// TIA Portal project "ODK_Test" (V14)

(* hardware
DEVICE "OC1"  CPU 1515SP PC
   slot 0: "OC1"  CPU 1515SP PC  6ES7 677-2AAxx-0xB0  V2.0
      slot 124: "Diagbase"  Diagbase  V6.0.4
      slot 125: "OC1"  PC Station 2.0  Station_Manager  V2.1
   slot 1: "CPU1505_v2"  CPU 1505SP  6ES7 672-5DC01-0YA0  V2.0
      slot 3: "CPU display_1"  6ES7591-1BA00-0AA0
   slot 2: "PROFINET onboard_2"  IE General  IE_CP  V2.1.0
   slot 127: "BA 2xRJ45"  BA 2xRJ45  6ES7 193-6AR00-0AA0  V0.0
      slot 32769: "Port_1"  6ES7 193-6AR00-0AA0
      slot 32770: "Port_2"  6ES7 193-6AR00-0AA0
   slot 1002: "Server module_1"  Server module  6ES7 193-6PA00-0AA0  V1.1
      slot 1: "Server module_1"  Server module
DEVICE "HMI_1"  KTP700 Basic PN
   slot 0: "KTP700 Basic PN"  KTP700 Basic PN  6AV2 123-2GB03-0AX0  14.0.0.0
   slot 1: "HMI_RT_1"  KTP700 Basic PN  6AV2 123-2GB03-0AX0  14.0.0.0
   slot 5: "HMI_1.IE_CP_1"  PROFINET Interface  14.0.0.0
      slot 1: "PROFINET Interface_1"  PROFINET Interface
         slot 1: "Port_1"  Port
*)

// ===== PLC "CPU1505_v2"  CPU 1505SP =====

VAR_GLOBAL   // PLC tag table "Default tag table"
   "System_Byte" AT %MB1 : Byte;
   "FirstScan" AT %M1.0 : Bool;
   "DiagStatusUpdate" AT %M1.1 : Bool;
   "AlwaysTRUE" AT %M1.2 : Bool;
   "AlwaysFALSE" AT %M1.3 : Bool;
   "Clock_Byte" AT %MB0 : Byte;
   "Clock_10Hz" AT %M0.0 : Bool;
   "Clock_5Hz" AT %M0.1 : Bool;
   "Clock_2.5Hz" AT %M0.2 : Bool;
   "Clock_2Hz" AT %M0.3 : Bool;
   "Clock_1.25Hz" AT %M0.4 : Bool;
   "Clock_1Hz" AT %M0.5 : Bool;
   "Clock_0.625Hz" AT %M0.6 : Bool;
   "Clock_0.5Hz" AT %M0.7 : Bool;
   "Tag_1" AT %M2.0 : Bool;
   "Tag_2" AT %M2.1 : Bool;
   "Tag_3" AT %M2.2 : Bool;
   "Tag_4" AT %M2.3 : Bool;
   "Tag_5" AT %M3.0 : Bool;
   "Tag_6" AT %M2.4 : Bool;
END_VAR

TYPE "FFT_Filter_RTComplex"
// This block is AUTO GENERATED - DO NOT MODIFY this block!
// Created by ODK_CodeGenerator version 200.0.3002.1
// at Sa Oktober 22 17:03:21 2016
// ********************************************************
   STRUCT
      re : Real;
      im : Real;
   END_STRUCT;
END_TYPE

DATA_BLOCK "FFT_Test_DB"   // DB1
{ S7_Optimized_Access := 'TRUE' }
VERSION : 0.1
// stored: InstanceOfName FFT_Test
"FFT_Test"
BEGIN
END_DATA_BLOCK

DATA_BLOCK "FFT_Filter_RT_Load_DB"   // DB2
{ S7_Optimized_Access := 'TRUE' }
VERSION : 0.1
// stored: InstanceOfName FFT_Filter_RT_Load
"FFT_Filter_RT_Load"
BEGIN
END_DATA_BLOCK

DATA_BLOCK "FFT_Filter_Params"   // DB3
{ S7_Optimized_Access := 'TRUE' }
VERSION : 0.1
   VAR
      FFT_Filter_Load : Struct
         Req_Press : Bool;
         Req : Bool;
         Done : Bool;
         Busy : Bool;
         Error : Bool;
         Status : Int;
      END_STRUCT;
      FFT_Filter_Unload : Struct
         Req_Press : Bool;
         Req : Bool;
         Done : Bool;
         Busy : Bool;
         Error : Bool;
         Status : Int;
      END_STRUCT;
      FFT_Data_Load : Struct
         Req_Press : Bool;
         Req : Bool;
         Done : Bool;
         Busy : Bool;
         Error : Bool;
         Status : Int;
      END_STRUCT;
      FFT_Data_Unload : Struct
         Req_Press : Bool;
         Req : Bool;
         Done : Bool;
         Busy : Bool;
         Error : Bool;
         Status : Int;
      END_STRUCT;
      FFT_Filter_Cycle : Struct
         FILT_EN : Bool;
         FILT_Status : Int;
         CycleDone : Bool;
         LastSample : Bool;
         CycleStartReq : Bool;
         CycleStartReqPress : Bool;
         CycleNumber : Int;
      END_STRUCT;
   END_VAR
BEGIN
END_DATA_BLOCK

DATA_BLOCK "FFT_Filter_RT_Unload_DB"   // DB4
{ S7_Optimized_Access := 'TRUE' }
VERSION : 0.1
// stored: InstanceOfName FFT_Filter_RT_Unload
"FFT_Filter_RT_Unload"
BEGIN
END_DATA_BLOCK

DATA_BLOCK "FFT_Filter_RTFFT1024p_DB"   // DB5
{ S7_Optimized_Access := 'TRUE' }
VERSION : 0.1
// stored: InstanceOfName FFT_Filter_RTFFT1024p
"FFT_Filter_RTFFT1024p"
BEGIN
END_DATA_BLOCK

DATA_BLOCK "FFT_Filter_RTFFT_Filt_DB"   // DB6
{ S7_Optimized_Access := 'TRUE' }
VERSION : 0.1
// stored: InstanceOfName FFT_Filter_RTFFT_Filt
"FFT_Filter_RTFFT_Filt"
BEGIN
END_DATA_BLOCK

DATA_BLOCK "FFT_Filter_RTLP_Filter_DB"   // DB7
{ S7_Optimized_Access := 'TRUE' }
VERSION : 0.1
// stored: InstanceOfName FFT_Filter_RTLP_Filter
"FFT_Filter_RTLP_Filter"
BEGIN
END_DATA_BLOCK

DATA_BLOCK "FFT_Filter_RTIFFT1024p_DB"   // DB8
{ S7_Optimized_Access := 'TRUE' }
VERSION : 0.1
// stored: InstanceOfName FFT_Filter_RTIFFT1024p
"FFT_Filter_RTIFFT1024p"
BEGIN
END_DATA_BLOCK

DATA_BLOCK "DataStreams"   // DB9
{ S7_Optimized_Access := 'TRUE' }
VERSION : 0.1
   VAR
      AudioCoefs_l_In : Array[0..1023] of Int;
      AudioCoefs_r_in : Array[0..1023] of Int;
      AudioCoefs_l_out : Array[0..1023] of Int;
      AudioCoefs_r_out : Array[0..1023] of Int;
   END_VAR
BEGIN
END_DATA_BLOCK

DATA_BLOCK "FFT_Filter_RTFFT_Filt_DB_1"   // DB10
{ S7_Optimized_Access := 'TRUE' }
VERSION : 0.1
// stored: InstanceOfName FFT_Filter_RTFFT_Filt
"FFT_Filter_RTFFT_Filt"
BEGIN
END_DATA_BLOCK

DATA_BLOCK "FFT_Filt_Data_Load_DB"   // DB11
{ S7_Optimized_Access := 'TRUE' }
VERSION : 0.1
// stored: InstanceOfName FFT_Filt_Data_Load
"FFT_Filt_Data_Load"
BEGIN
END_DATA_BLOCK

DATA_BLOCK "FFT_Filt_Data_Unload_DB"   // DB12
{ S7_Optimized_Access := 'TRUE' }
VERSION : 0.1
// stored: InstanceOfName FFT_Filt_Data_Unload
"FFT_Filt_Data_Unload"
BEGIN
END_DATA_BLOCK

DATA_BLOCK "FFT_Filt_DataWaveSetup_DB"   // DB13
{ S7_Optimized_Access := 'TRUE' }
VERSION : 0.1
// stored: InstanceOfName FFT_Filt_DataWaveSetup
"FFT_Filt_DataWaveSetup"
BEGIN
END_DATA_BLOCK

DATA_BLOCK "FFT_Filt_DataGetSamplesStereo_DB"   // DB14
{ S7_Optimized_Access := 'TRUE' }
VERSION : 0.1
// stored: InstanceOfName FFT_Filt_DataGetSamplesStereo
"FFT_Filt_DataGetSamplesStereo"
BEGIN
END_DATA_BLOCK

DATA_BLOCK "FFT_Filt_DataWriteSamples_DB"   // DB15
{ S7_Optimized_Access := 'TRUE' }
VERSION : 0.1
// stored: InstanceOfName FFT_Filt_DataWriteSamples
"FFT_Filt_DataWriteSamples"
BEGIN
END_DATA_BLOCK

FUNCTION_BLOCK "FFT_Filter_RT_Load"   // FB1, SCL
{ S7_Optimized_Access := 'TRUE' }
VERSION : 0.1
// This block is AUTO GENERATED - DO NOT MODIFY this block!
// Created by ODK_CodeGenerator version 200.0.3002.1
// at Sa Oktober 22 17:03:21 2016
// max. number of parallel calls into this ODK application is: 3
// *************************************************************
   VAR_INPUT
      REQ : Bool;
   END_VAR
   VAR_OUTPUT
      DONE : Bool;
      BUSY : Bool;
      ERROR : Bool;
      STATUS : Int;
   END_VAR
   VAR
      ODK_Load_Instance : ODK_Load;
      _odk_internal_LIBRARY_NAME : String := '<rt>FFT_Filter_RT.so';
   END_VAR
   VAR CONSTANT
      _odk_internal_INSTANCE_ID : UDInt := 1_300_268_953;
   END_VAR
BEGIN
   //
   // DO NOT CHANGE BELOW OF THIS LINE !!
   // This is an automatic generated block by the
   // SIMATIC ODK 1500S V2.0
   // DO NOT CHANGE !!
   //
   #ODK_Load_Instance(REQ := #REQ,
                      LIBRARY_NAME := #_odk_internal_LIBRARY_NAME,
                      INSTANCE_ID := #_odk_internal_INSTANCE_ID,
                      DONE => #DONE,
                      BUSY => #BUSY,
                      ERROR => #ERROR,
                      STATUS => #STATUS);
   //
   // DO NOT CHANGE !!
   // This is an automatic generated block by the
   // SIMATIC ODK 1500S V2.0
   // DO NOT CHANGE ABOVE OF THIS LINE !!
   //
END_FUNCTION_BLOCK

FUNCTION_BLOCK "FFT_Filter_RT_Unload"   // FB2, SCL
{ S7_Optimized_Access := 'TRUE' }
VERSION : 0.1
// This block is AUTO GENERATED - DO NOT MODIFY this block!
// Created by ODK_CodeGenerator version 200.0.3002.1
// at Sa Oktober 22 17:03:21 2016
// max. number of parallel calls into this ODK application is: 3
// *************************************************************
   VAR_INPUT
      REQ : Bool;
   END_VAR
   VAR_OUTPUT
      DONE : Bool;
      BUSY : Bool;
      ERROR : Bool;
      STATUS : Int;
   END_VAR
   VAR
      ODK_Unld_Instance : ODK_Unld;
   END_VAR
   VAR CONSTANT
      _odk_internal_INSTANCE_ID : UDInt := 1_300_268_953;
   END_VAR
BEGIN
   //
   // DO NOT CHANGE BELOW OF THIS LINE !!
   // This is an automatic generated block by the
   // SIMATIC ODK 1500S V2.0
   // DO NOT CHANGE !!
   //
   #ODK_Unld_Instance(REQ := #REQ,
                      INSTANCE_ID := #_odk_internal_INSTANCE_ID,
                      DONE => #DONE,
                      BUSY => #BUSY,
                      ERROR => #ERROR,
                      STATUS => #STATUS);
   //
   // DO NOT CHANGE !!
   // This is an automatic generated block by the
   // SIMATIC ODK 1500S V2.0
   // DO NOT CHANGE ABOVE OF THIS LINE !!
   //
END_FUNCTION_BLOCK

FUNCTION_BLOCK "FFT_Filter_RTFFT1024p"   // FB3, SCL
{ S7_Optimized_Access := 'TRUE' }
VERSION : 0.1
// This block is AUTO GENERATED - DO NOT MODIFY this block!
// Created by ODK_CodeGenerator version 200.0.3002.1
// at Sa Oktober 22 17:03:21 2016
// max. number of parallel calls into this ODK application is: 3
// *************************************************************
//  perform a 1024 point fast fourier transformation
   VAR_INPUT
      timeCoef : Array[0..1023] of Int;   // time domain coefficients
   END_VAR
   VAR_OUTPUT
      STATUS : Int := 0;
      freqCoef : Array[0..1023] of "FFT_Filter_RTComplex";   // frequency domain coefficients
   END_VAR
   VAR
      _odk_internal_Last_REQ : Bool := FALSE;
      _odk_internal_Last_BUSY : Bool := FALSE;
      _odk_internal_IN_BUFFER : Array[0..2047] of Byte;
      _odk_internal_OUT_BUFFER : Array[0..8191] of Byte;
   END_VAR
   VAR_TEMP
      _odk_internal_pos : DInt;
      _odk_internal_err : Int;
      _odk_internal_i : Int;
      _odk_internal_udt_0 : Int;
   END_VAR
   VAR CONSTANT
      _odk_internal_INSTANCE_ID : UDInt := 1_300_268_953;
      _odk_internal_COMMAND : UDInt := 3_762_803_041;
   END_VAR
BEGIN
   //
   // DO NOT CHANGE BELOW OF THIS LINE !!
   // This is an automatic generated block by the
   // SIMATIC ODK 1500S V2.0
   // DO NOT CHANGE !!
   //
   // perform a 1024 point fast fourier transformation                       
   #_odk_internal_pos := 0;
   FOR #_odk_internal_i := 0 TO 1023 DO
       #_odk_internal_err := WRITE_LITTLE(src_variable := #timeCoef[#_odk_internal_i], dest_array := #_odk_internal_IN_BUFFER, pos := #_odk_internal_pos);
   END_FOR;
   #STATUS := ODK_ExcS(INSTANCE_ID := #_odk_internal_INSTANCE_ID,
                       COMMAND := #_odk_internal_COMMAND,
                       IN_DATA := #_odk_internal_IN_BUFFER,
                       INOUT_DATA := null,
                       OUT_DATA := #_odk_internal_OUT_BUFFER
   );
   IF INT_TO_UINT(#STATUS) < 16#7000 THEN
       #_odk_internal_pos := 0;
       FOR #_odk_internal_udt_0 := 0 TO 1023 DO
           #_odk_internal_err := READ_LITTLE(dest_Variable => #freqCoef[#_odk_internal_udt_0].re, src_array := #_odk_internal_OUT_BUFFER, pos := #_odk_internal_pos);
           #_odk_internal_err := READ_LITTLE(dest_Variable => #freqCoef[#_odk_internal_udt_0].im, src_array := #_odk_internal_OUT_BUFFER, pos := #_odk_internal_pos);
       END_FOR;
   END_IF;
   //
   // DO NOT CHANGE !!
   // This is an automatic generated block by the
   // SIMATIC ODK 1500S V2.0
   // DO NOT CHANGE ABOVE OF THIS LINE !!
   //
END_FUNCTION_BLOCK

FUNCTION_BLOCK "FFT_Filter_RTLP_Filter"   // FB4, SCL
{ S7_Optimized_Access := 'TRUE' }
VERSION : 0.1
// This block is AUTO GENERATED - DO NOT MODIFY this block!
// Created by ODK_CodeGenerator version 200.0.3002.1
// at Sa Oktober 22 17:03:21 2016
// max. number of parallel calls into this ODK application is: 3
// *************************************************************
//  multiply complex coeffs with a filter function
   VAR_INPUT
      freqCoef : Array[0..1023] of "FFT_Filter_RTComplex";   // filter input
   END_VAR
   VAR_OUTPUT
      STATUS : Int := 0;
      freqCoefFilt : Array[0..1023] of "FFT_Filter_RTComplex";   // filter output
   END_VAR
   VAR
      _odk_internal_Last_REQ : Bool := FALSE;
      _odk_internal_Last_BUSY : Bool := FALSE;
      _odk_internal_IN_BUFFER : Array[0..8191] of Byte;
      _odk_internal_OUT_BUFFER : Array[0..8191] of Byte;
   END_VAR
   VAR_TEMP
      _odk_internal_pos : DInt;
      _odk_internal_err : Int;
      _odk_internal_i : Int;
      _odk_internal_udt_0 : Int;
   END_VAR
   VAR CONSTANT
      _odk_internal_INSTANCE_ID : UDInt := 1_300_268_953;
      _odk_internal_COMMAND : UDInt := 1_993_759_514;
   END_VAR
BEGIN
   //
   // DO NOT CHANGE BELOW OF THIS LINE !!
   // This is an automatic generated block by the
   // SIMATIC ODK 1500S V2.0
   // DO NOT CHANGE !!
   //
   // multiply complex coeffs with a filter function                        
   #_odk_internal_pos := 0;
   FOR #_odk_internal_udt_0 := 0 TO 1023 DO
       #_odk_internal_err := WRITE_LITTLE(src_variable := #freqCoef[#_odk_internal_udt_0].re, dest_array := #_odk_internal_IN_BUFFER, pos := #_odk_internal_pos);
       #_odk_internal_err := WRITE_LITTLE(src_variable := #freqCoef[#_odk_internal_udt_0].im, dest_array := #_odk_internal_IN_BUFFER, pos := #_odk_internal_pos);
   END_FOR;
   #STATUS := ODK_ExcS(INSTANCE_ID := #_odk_internal_INSTANCE_ID,
                       COMMAND := #_odk_internal_COMMAND,
                       IN_DATA := #_odk_internal_IN_BUFFER,
                       INOUT_DATA := null,
                       OUT_DATA := #_odk_internal_OUT_BUFFER
   );
   IF INT_TO_UINT(#STATUS) < 16#7000 THEN
       #_odk_internal_pos := 0;
       FOR #_odk_internal_udt_0 := 0 TO 1023 DO
           #_odk_internal_err := READ_LITTLE(dest_Variable => #freqCoefFilt[#_odk_internal_udt_0].re, src_array := #_odk_internal_OUT_BUFFER, pos := #_odk_internal_pos);
           #_odk_internal_err := READ_LITTLE(dest_Variable => #freqCoefFilt[#_odk_internal_udt_0].im, src_array := #_odk_internal_OUT_BUFFER, pos := #_odk_internal_pos);
       END_FOR;
   END_IF;
   //
   // DO NOT CHANGE !!
   // This is an automatic generated block by the
   // SIMATIC ODK 1500S V2.0
   // DO NOT CHANGE ABOVE OF THIS LINE !!
   //
END_FUNCTION_BLOCK

FUNCTION_BLOCK "FFT_Filter_RTIFFT1024p"   // FB5, SCL
{ S7_Optimized_Access := 'TRUE' }
VERSION : 0.1
// This block is AUTO GENERATED - DO NOT MODIFY this block!
// Created by ODK_CodeGenerator version 200.0.3002.1
// at Sa Oktober 22 17:03:21 2016
// max. number of parallel calls into this ODK application is: 3
// *************************************************************
//  perform an inverse 1024 point fast fourier transformation
   VAR_INPUT
      freqCoef : Array[0..1023] of "FFT_Filter_RTComplex";   // frequency domain coefficients
   END_VAR
   VAR_OUTPUT
      STATUS : Int := 0;
      timeCoefOut : Array[0..1023] of Int;   // time domain coefficients
   END_VAR
   VAR
      _odk_internal_Last_REQ : Bool := FALSE;
      _odk_internal_Last_BUSY : Bool := FALSE;
      _odk_internal_IN_BUFFER : Array[0..8191] of Byte;
      _odk_internal_OUT_BUFFER : Array[0..2047] of Byte;
   END_VAR
   VAR_TEMP
      _odk_internal_pos : DInt;
      _odk_internal_err : Int;
      _odk_internal_i : Int;
      _odk_internal_udt_0 : Int;
   END_VAR
   VAR CONSTANT
      _odk_internal_INSTANCE_ID : UDInt := 1_300_268_953;
      _odk_internal_COMMAND : UDInt := 93215674;
   END_VAR
BEGIN
   //
   // DO NOT CHANGE BELOW OF THIS LINE !!
   // This is an automatic generated block by the
   // SIMATIC ODK 1500S V2.0
   // DO NOT CHANGE !!
   //
   // perform an inverse 1024 point fast fourier transformation                   
   #_odk_internal_pos := 0;
   FOR #_odk_internal_udt_0 := 0 TO 1023 DO
       #_odk_internal_err := WRITE_LITTLE(src_variable := #freqCoef[#_odk_internal_udt_0].re, dest_array := #_odk_internal_IN_BUFFER, pos := #_odk_internal_pos);
       #_odk_internal_err := WRITE_LITTLE(src_variable := #freqCoef[#_odk_internal_udt_0].im, dest_array := #_odk_internal_IN_BUFFER, pos := #_odk_internal_pos);
   END_FOR;
   #STATUS := ODK_ExcS(INSTANCE_ID := #_odk_internal_INSTANCE_ID,
                       COMMAND := #_odk_internal_COMMAND,
                       IN_DATA := #_odk_internal_IN_BUFFER,
                       INOUT_DATA := null,
                       OUT_DATA := #_odk_internal_OUT_BUFFER
   );
   IF INT_TO_UINT(#STATUS) < 16#7000 THEN
       #_odk_internal_pos := 0;
       FOR #_odk_internal_i := 0 TO 1023 DO
           #_odk_internal_err := READ_LITTLE(dest_Variable => #timeCoefOut[#_odk_internal_i], src_array := #_odk_internal_OUT_BUFFER, pos := #_odk_internal_pos);
       END_FOR;
   END_IF;
   //
   // DO NOT CHANGE !!
   // This is an automatic generated block by the
   // SIMATIC ODK 1500S V2.0
   // DO NOT CHANGE ABOVE OF THIS LINE !!
   //
END_FUNCTION_BLOCK

FUNCTION_BLOCK "FFT_Filter_RTFFT_Filt"   // FB6, SCL
{ S7_Optimized_Access := 'TRUE' }
VERSION : 0.1
// This block is AUTO GENERATED - DO NOT MODIFY this block!
// Created by ODK_CodeGenerator version 200.0.3002.1
// at Sa Oktober 22 17:03:21 2016
// max. number of parallel calls into this ODK application is: 3
// *************************************************************
//  perform a full filter with FFT->Filter->IFFT
   VAR_INPUT
      timeCoef : Array[0..1023] of Int;   // time domain input coefficients
   END_VAR
   VAR_OUTPUT
      STATUS : Int := 0;
      timeCoefOut : Array[0..1023] of Int;   // time domain output coefficients
   END_VAR
   VAR
      _odk_internal_Last_REQ : Bool := FALSE;
      _odk_internal_Last_BUSY : Bool := FALSE;
      _odk_internal_IN_BUFFER : Array[0..2047] of Byte;
      _odk_internal_OUT_BUFFER : Array[0..2047] of Byte;
   END_VAR
   VAR_TEMP
      _odk_internal_pos : DInt;
      _odk_internal_err : Int;
      _odk_internal_i : Int;
   END_VAR
   VAR CONSTANT
      _odk_internal_INSTANCE_ID : UDInt := 1_300_268_953;
      _odk_internal_COMMAND : UDInt := 1_847_992_643;
   END_VAR
BEGIN
   //
   // DO NOT CHANGE BELOW OF THIS LINE !!
   // This is an automatic generated block by the
   // SIMATIC ODK 1500S V2.0
   // DO NOT CHANGE !!
   //
   // perform a full filter with FFT->Filter->IFFT
   #_odk_internal_pos := 0;
   FOR #_odk_internal_i := 0 TO 1023 DO
       #_odk_internal_err := WRITE_LITTLE(src_variable := #timeCoef[#_odk_internal_i], dest_array := #_odk_internal_IN_BUFFER, pos := #_odk_internal_pos);
   END_FOR;
   #STATUS := ODK_ExcS(INSTANCE_ID := #_odk_internal_INSTANCE_ID,
                       COMMAND := #_odk_internal_COMMAND,
                       IN_DATA := #_odk_internal_IN_BUFFER,
                       INOUT_DATA := null,
                       OUT_DATA := #_odk_internal_OUT_BUFFER
   );
   IF INT_TO_UINT(#STATUS) < 16#7000 THEN
       #_odk_internal_pos := 0;
       FOR #_odk_internal_i := 0 TO 1023 DO
           #_odk_internal_err := READ_LITTLE(dest_Variable => #timeCoefOut[#_odk_internal_i], src_array := #_odk_internal_OUT_BUFFER, pos := #_odk_internal_pos);
       END_FOR;
   END_IF;
   //
   // DO NOT CHANGE !!
   // This is an automatic generated block by the
   // SIMATIC ODK 1500S V2.0
   // DO NOT CHANGE ABOVE OF THIS LINE !!
   //
END_FUNCTION_BLOCK

FUNCTION_BLOCK "FFT_Filter_RT_GetTrace"   // FB7, SCL
{ S7_Optimized_Access := 'TRUE' }
VERSION : 0.1
// This block is AUTO GENERATED - DO NOT MODIFY this block!
// Created by ODK_CodeGenerator version 200.0.3002.1
// at Sa Oktober 22 17:03:21 2016
// max. number of parallel calls into this ODK application is: 3
// *************************************************************
   VAR_INPUT
      TraceCount : Int;
   END_VAR
   VAR_OUTPUT
      STATUS : Int := 0;
      TraceBuffer : Array[0..255] of String[125];
   END_VAR
   VAR
      _odk_internal_Last_REQ : Bool := FALSE;
      _odk_internal_Last_BUSY : Bool := FALSE;
      _odk_internal_IN_BUFFER : Array[0..1] of Byte;
      _odk_internal_OUT_BUFFER : Array[0..32511] of Byte;
   END_VAR
   VAR_TEMP
      _odk_internal_pos : DInt;
      _odk_internal_err : Int;
      _odk_internal_i : Int;
      _odk_internal_tmpStringLen : Byte;
      _odk_internal_j : Int;
      _odk_internal_tmp_string : String;
   END_VAR
   VAR CONSTANT
      _odk_internal_INSTANCE_ID : UDInt := 1_300_268_953;
      _odk_internal_COMMAND : UDInt := 4_033_566_251;
   END_VAR
BEGIN
   //
   // DO NOT CHANGE BELOW OF THIS LINE !!
   // This is an automatic generated block by the
   // SIMATIC ODK 1500S V2.0
   // DO NOT CHANGE !!
   //
   #_odk_internal_pos := 0;
   #_odk_internal_err := WRITE_LITTLE(src_variable := #TraceCount, dest_array := #_odk_internal_IN_BUFFER, pos := #_odk_internal_pos);
   #STATUS := ODK_ExcS(INSTANCE_ID := #_odk_internal_INSTANCE_ID,
                       COMMAND := #_odk_internal_COMMAND,
                       IN_DATA := #_odk_internal_IN_BUFFER,
                       INOUT_DATA := null,
                       OUT_DATA := #_odk_internal_OUT_BUFFER
   );
   IF INT_TO_UINT(#STATUS) < 16#7000 THEN
       #_odk_internal_pos := 0;
       FOR #_odk_internal_j := 0 TO 255 DO
           #_odk_internal_tmp_string := '';
           #_odk_internal_tmpStringLen := #_odk_internal_OUT_BUFFER[#_odk_internal_pos];
           #_odk_internal_pos := #_odk_internal_pos + 1;
           #_odk_internal_tmpStringLen := #_odk_internal_OUT_BUFFER[#_odk_internal_pos];
           #_odk_internal_pos := #_odk_internal_pos + 1;
           FOR #_odk_internal_i := 1 TO BYTE_TO_INT(#_odk_internal_tmpStringLen) DO
               #_odk_internal_tmp_string[#_odk_internal_i] := BYTE_TO_CHAR(#_odk_internal_OUT_BUFFER[#_odk_internal_pos]);
               #_odk_internal_pos := #_odk_internal_pos + 1;
           END_FOR;
           #_odk_internal_pos := #_odk_internal_pos + 125 - LEN(#_odk_internal_tmp_string);
           #TraceBuffer[#_odk_internal_j] := #_odk_internal_tmp_string;
       END_FOR;
   END_IF;
   //
   // DO NOT CHANGE !!
   // This is an automatic generated block by the
   // SIMATIC ODK 1500S V2.0
   // DO NOT CHANGE ABOVE OF THIS LINE !!
   //
END_FUNCTION_BLOCK

FUNCTION_BLOCK "FFT_Test"   // FB8, FBD
{ S7_Optimized_Access := 'TRUE' }
VERSION : 0.1
BEGIN

REGION Network 1: Load and Unload
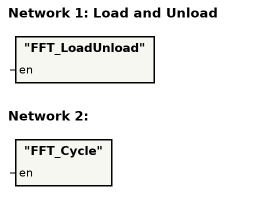
   "FFT_LoadUnload"();
END_REGION

REGION Network 2
   "FFT_Cycle"();
END_REGION
END_FUNCTION_BLOCK

FUNCTION_BLOCK "FFT_Filt_Data_Load"   // FB9, SCL
{ S7_Optimized_Access := 'TRUE' }
VERSION : 0.1
// This block is AUTO GENERATED - DO NOT MODIFY this block!
// Created by ODK_CodeGenerator version 200.0.3002.1
// at Sa Oktober 22 17:12:18 2016
// ********************************************************
   VAR_INPUT
      REQ : Bool;
   END_VAR
   VAR_OUTPUT
      DONE : Bool;
      BUSY : Bool;
      ERROR : Bool;
      STATUS : Int;
   END_VAR
   VAR
      ODK_Load_Instance : ODK_Load;
      _odk_internal_LIBRARY_NAME : String := '<nrt>FFT_Filt_Data.dll';
   END_VAR
   VAR CONSTANT
      _odk_internal_INSTANCE_ID : UDInt := 4_055_393_781;
   END_VAR
BEGIN
   //
   // DO NOT CHANGE BELOW OF THIS LINE !!
   // This is an automatic generated block by the
   // SIMATIC ODK 1500S V2.0
   // DO NOT CHANGE !!
   //
   #ODK_Load_Instance(REQ := #REQ,
                      LIBRARY_NAME := #_odk_internal_LIBRARY_NAME,
                      INSTANCE_ID := #_odk_internal_INSTANCE_ID,
                      DONE => #DONE,
                      BUSY => #BUSY,
                      ERROR => #ERROR,
                      STATUS => #STATUS);
   //
   // DO NOT CHANGE !!
   // This is an automatic generated block by the
   // SIMATIC ODK 1500S V2.0
   // DO NOT CHANGE ABOVE OF THIS LINE !!
   //
END_FUNCTION_BLOCK

FUNCTION_BLOCK "FFT_Filt_Data_Unload"   // FB10, SCL
{ S7_Optimized_Access := 'TRUE' }
VERSION : 0.1
// This block is AUTO GENERATED - DO NOT MODIFY this block!
// Created by ODK_CodeGenerator version 200.0.3002.1
// at Sa Oktober 22 17:12:18 2016
// ********************************************************
   VAR_INPUT
      REQ : Bool;
   END_VAR
   VAR_OUTPUT
      DONE : Bool;
      BUSY : Bool;
      ERROR : Bool;
      STATUS : Int;
   END_VAR
   VAR
      ODK_Unld_Instance : ODK_Unld;
   END_VAR
   VAR CONSTANT
      _odk_internal_INSTANCE_ID : UDInt := 4_055_393_781;
   END_VAR
BEGIN
   //
   // DO NOT CHANGE BELOW OF THIS LINE !!
   // This is an automatic generated block by the
   // SIMATIC ODK 1500S V2.0
   // DO NOT CHANGE !!
   //
   #ODK_Unld_Instance(REQ := #REQ,
                      INSTANCE_ID := #_odk_internal_INSTANCE_ID,
                      DONE => #DONE,
                      BUSY => #BUSY,
                      ERROR => #ERROR,
                      STATUS => #STATUS);
   //
   // DO NOT CHANGE !!
   // This is an automatic generated block by the
   // SIMATIC ODK 1500S V2.0
   // DO NOT CHANGE ABOVE OF THIS LINE !!
   //
END_FUNCTION_BLOCK

FUNCTION_BLOCK "FFT_Filt_DataWaveSetup"   // FB11, SCL
{ S7_Optimized_Access := 'TRUE' }
VERSION : 0.1
// This block is AUTO GENERATED - DO NOT MODIFY this block!
// Created by ODK_CodeGenerator version 200.0.3002.1
// at Sa Oktober 22 17:12:18 2016
// ********************************************************
//  Setup file handles for IO operation
   VAR_INPUT
      REQ : Bool;
      inFileName : String[254];   // input wave
      outFileName : String[254];   // output to write to
   END_VAR
   VAR_OUTPUT
      ERROR : Bool := FALSE;
      DONE : Bool := FALSE;
      BUSY : Bool := FALSE;
      STATUS : Int := 0;
   END_VAR
   VAR
      _odk_internal_Last_REQ : Bool := FALSE;
      _odk_internal_Last_BUSY : Bool := FALSE;
      ODK_ExcA_Instance : ODK_ExcA;
      _odk_internal_IN_BUFFER : Array[0..511] of Byte;
   END_VAR
   VAR_TEMP
      _odk_internal_pos : DInt;
      _odk_internal_err : Int;
      _odk_internal_i : Int;
      _odk_internal_tmpStringLen : Byte;
   END_VAR
   VAR CONSTANT
      _odk_internal_INSTANCE_ID : UDInt := 4_055_393_781;
      _odk_internal_COMMAND : UDInt := 2_806_550_197;
   END_VAR
BEGIN
   //
   // DO NOT CHANGE BELOW OF THIS LINE !!
   // This is an automatic generated block by the
   // SIMATIC ODK 1500S V2.0
   // DO NOT CHANGE !!
   //
   // Setup file handles for IO operation
   IF NOT #_odk_internal_Last_REQ & #REQ & NOT #_odk_internal_Last_BUSY THEN
       #_odk_internal_pos := 0;
       #_odk_internal_tmpStringLen := INT_TO_BYTE(LEN(#inFileName));
       #_odk_internal_IN_BUFFER[#_odk_internal_pos] := BYTE#254;
       #_odk_internal_pos := #_odk_internal_pos + 1;
       #_odk_internal_IN_BUFFER[#_odk_internal_pos] := #_odk_internal_tmpStringLen;
       #_odk_internal_pos := #_odk_internal_pos + 1;
       FOR #_odk_internal_i := 1 TO BYTE_TO_INT(#_odk_internal_tmpStringLen) DO
           #_odk_internal_IN_BUFFER[#_odk_internal_pos] := CHAR_TO_BYTE(#inFileName[#_odk_internal_i]);
           #_odk_internal_pos := #_odk_internal_pos + 1;
       END_FOR;
       #_odk_internal_pos := #_odk_internal_pos + 254 - #_odk_internal_tmpStringLen;
       #_odk_internal_tmpStringLen := INT_TO_BYTE(LEN(#outFileName));
       #_odk_internal_IN_BUFFER[#_odk_internal_pos] := BYTE#254;
       #_odk_internal_pos := #_odk_internal_pos + 1;
       #_odk_internal_IN_BUFFER[#_odk_internal_pos] := #_odk_internal_tmpStringLen;
       #_odk_internal_pos := #_odk_internal_pos + 1;
       FOR #_odk_internal_i := 1 TO BYTE_TO_INT(#_odk_internal_tmpStringLen) DO
           #_odk_internal_IN_BUFFER[#_odk_internal_pos] := CHAR_TO_BYTE(#outFileName[#_odk_internal_i]);
           #_odk_internal_pos := #_odk_internal_pos + 1;
       END_FOR;
       #_odk_internal_pos := #_odk_internal_pos + 254 - #_odk_internal_tmpStringLen;

   END_IF;
   #_odk_internal_Last_REQ := #REQ;
   #ODK_ExcA_Instance(REQ := #REQ,
                      INSTANCE_ID := #_odk_internal_INSTANCE_ID,
                      COMMAND := #_odk_internal_COMMAND,
                      IN_DATA := #_odk_internal_IN_BUFFER,
                      INOUT_DATA := null,
                      OUT_DATA := null,
                      DONE => #DONE,
                      BUSY => #BUSY,
                      ERROR => #ERROR,
                      STATUS => #STATUS);
   #_odk_internal_Last_BUSY := #BUSY;
   //
   // DO NOT CHANGE !!
   // This is an automatic generated block by the
   // SIMATIC ODK 1500S V2.0
   // DO NOT CHANGE ABOVE OF THIS LINE !!
   //
END_FUNCTION_BLOCK

FUNCTION_BLOCK "FFT_Filt_DataWaveSetupNoName"   // FB12, SCL
{ S7_Optimized_Access := 'TRUE' }
VERSION : 0.1
// This block is AUTO GENERATED - DO NOT MODIFY this block!
// Created by ODK_CodeGenerator version 200.0.3002.1
// at Sa Oktober 22 17:12:18 2016
// ********************************************************
//  Test Setup file handles without name
   VAR_INPUT
      REQ : Bool;
   END_VAR
   VAR_OUTPUT
      ERROR : Bool := FALSE;
      DONE : Bool := FALSE;
      BUSY : Bool := FALSE;
      STATUS : Int := 0;
   END_VAR
   VAR
      _odk_internal_Last_REQ : Bool := FALSE;
      _odk_internal_Last_BUSY : Bool := FALSE;
      ODK_ExcA_Instance : ODK_ExcA;
   END_VAR
   VAR_TEMP
      _odk_internal_pos : DInt;
      _odk_internal_err : Int;
      _odk_internal_i : Int;
   END_VAR
   VAR CONSTANT
      _odk_internal_INSTANCE_ID : UDInt := 4_055_393_781;
      _odk_internal_COMMAND : UDInt := 1_271_720_052;
   END_VAR
BEGIN
   //
   // DO NOT CHANGE BELOW OF THIS LINE !!
   // This is an automatic generated block by the
   // SIMATIC ODK 1500S V2.0
   // DO NOT CHANGE !!
   //
   // Test Setup file handles without name
   #_odk_internal_Last_REQ := #REQ;
   #ODK_ExcA_Instance(REQ := #REQ,
                      INSTANCE_ID := #_odk_internal_INSTANCE_ID,
                      COMMAND := #_odk_internal_COMMAND,
                      IN_DATA := null,
                      INOUT_DATA := null,
                      OUT_DATA := null,
                      DONE => #DONE,
                      BUSY => #BUSY,
                      ERROR => #ERROR,
                      STATUS => #STATUS);
   #_odk_internal_Last_BUSY := #BUSY;
   //
   // DO NOT CHANGE !!
   // This is an automatic generated block by the
   // SIMATIC ODK 1500S V2.0
   // DO NOT CHANGE ABOVE OF THIS LINE !!
   //
END_FUNCTION_BLOCK

FUNCTION_BLOCK "FFT_Filt_DataGetSamplesStereo"   // FB13, SCL
{ S7_Optimized_Access := 'TRUE' }
VERSION : 0.1
// This block is AUTO GENERATED - DO NOT MODIFY this block!
// Created by ODK_CodeGenerator version 200.0.3002.1
// at Sa Oktober 22 17:12:18 2016
// ********************************************************
//  Get one filter samlple for processing
   VAR_INPUT
      REQ : Bool;
   END_VAR
   VAR_OUTPUT
      ERROR : Bool := FALSE;
      DONE : Bool := FALSE;
      BUSY : Bool := FALSE;
      STATUS : Int := 0;
      inputSamplesL : Array[0..1023] of Int;   // input audio samples left
      inputSamplesR : Array[0..1023] of Int;   // input audio samples right
      lastSample : Bool;   // last sample indicator
   END_VAR
   VAR
      _odk_internal_Last_REQ : Bool := FALSE;
      _odk_internal_Last_BUSY : Bool := FALSE;
      ODK_ExcA_Instance : ODK_ExcA;
      _odk_internal_OUT_BUFFER : Array[0..4096] of Byte;
   END_VAR
   VAR_TEMP
      _odk_internal_pos : DInt;
      _odk_internal_err : Int;
      _odk_internal_i : Int;
   END_VAR
   VAR CONSTANT
      _odk_internal_INSTANCE_ID : UDInt := 4_055_393_781;
      _odk_internal_COMMAND : UDInt := 2_530_698_148;
   END_VAR
BEGIN
   //
   // DO NOT CHANGE BELOW OF THIS LINE !!
   // This is an automatic generated block by the
   // SIMATIC ODK 1500S V2.0
   // DO NOT CHANGE !!
   //
   // Get one filter samlple for processing   
   #_odk_internal_Last_REQ := #REQ;
   #ODK_ExcA_Instance(REQ := #REQ,
                      INSTANCE_ID := #_odk_internal_INSTANCE_ID,
                      COMMAND := #_odk_internal_COMMAND,
                      IN_DATA := null,
                      INOUT_DATA := null,
                      OUT_DATA := #_odk_internal_OUT_BUFFER,
                      DONE => #DONE,
                      BUSY => #BUSY,
                      ERROR => #ERROR,
                      STATUS => #STATUS);
   IF NOT #BUSY & #_odk_internal_Last_BUSY & NOT #ERROR THEN
       #_odk_internal_pos := 0;
       FOR #_odk_internal_i := 0 TO 1023 DO
           #_odk_internal_err := READ_LITTLE(dest_Variable => #inputSamplesL[#_odk_internal_i], src_array := #_odk_internal_OUT_BUFFER, pos := #_odk_internal_pos);
       END_FOR;
       FOR #_odk_internal_i := 0 TO 1023 DO
           #_odk_internal_err := READ_LITTLE(dest_Variable => #inputSamplesR[#_odk_internal_i], src_array := #_odk_internal_OUT_BUFFER, pos := #_odk_internal_pos);
       END_FOR;
       #lastSample := BYTE_TO_BOOL(#_odk_internal_OUT_BUFFER[#_odk_internal_pos]);
       #_odk_internal_pos := #_odk_internal_pos + 1;
   END_IF;
   #_odk_internal_Last_BUSY := #BUSY;
   //
   // DO NOT CHANGE !!
   // This is an automatic generated block by the
   // SIMATIC ODK 1500S V2.0
   // DO NOT CHANGE ABOVE OF THIS LINE !!
   //
END_FUNCTION_BLOCK

FUNCTION_BLOCK "FFT_Filt_DataWriteSamples"   // FB14, SCL
{ S7_Optimized_Access := 'TRUE' }
VERSION : 0.1
// This block is AUTO GENERATED - DO NOT MODIFY this block!
// Created by ODK_CodeGenerator version 200.0.3002.1
// at Sa Oktober 22 17:12:18 2016
// ********************************************************
//  write processed sample frame into file
   VAR_INPUT
      REQ : Bool;
      filteredSamplesL : Array[0..1023] of Int;   // output to write to left chan
      filteredSamplesR : Array[0..1023] of Int;   // output to write to right chan
   END_VAR
   VAR_OUTPUT
      ERROR : Bool := FALSE;
      DONE : Bool := FALSE;
      BUSY : Bool := FALSE;
      STATUS : Int := 0;
   END_VAR
   VAR
      _odk_internal_Last_REQ : Bool := FALSE;
      _odk_internal_Last_BUSY : Bool := FALSE;
      ODK_ExcA_Instance : ODK_ExcA;
      _odk_internal_IN_BUFFER : Array[0..4095] of Byte;
   END_VAR
   VAR_TEMP
      _odk_internal_pos : DInt;
      _odk_internal_err : Int;
      _odk_internal_i : Int;
   END_VAR
   VAR CONSTANT
      _odk_internal_INSTANCE_ID : UDInt := 4_055_393_781;
      _odk_internal_COMMAND : UDInt := 1_897_094_642;
   END_VAR
BEGIN
   //
   // DO NOT CHANGE BELOW OF THIS LINE !!
   // This is an automatic generated block by the
   // SIMATIC ODK 1500S V2.0
   // DO NOT CHANGE !!
   //
   // write processed sample frame into file
   IF NOT #_odk_internal_Last_REQ & #REQ & NOT #_odk_internal_Last_BUSY THEN
       #_odk_internal_pos := 0;
       FOR #_odk_internal_i := 0 TO 1023 DO
           #_odk_internal_err := WRITE_LITTLE(src_variable := #filteredSamplesL[#_odk_internal_i], dest_array := #_odk_internal_IN_BUFFER, pos := #_odk_internal_pos);
       END_FOR;
       FOR #_odk_internal_i := 0 TO 1023 DO
           #_odk_internal_err := WRITE_LITTLE(src_variable := #filteredSamplesR[#_odk_internal_i], dest_array := #_odk_internal_IN_BUFFER, pos := #_odk_internal_pos);
       END_FOR;

   END_IF;
   #_odk_internal_Last_REQ := #REQ;
   #ODK_ExcA_Instance(REQ := #REQ,
                      INSTANCE_ID := #_odk_internal_INSTANCE_ID,
                      COMMAND := #_odk_internal_COMMAND,
                      IN_DATA := #_odk_internal_IN_BUFFER,
                      INOUT_DATA := null,
                      OUT_DATA := null,
                      DONE => #DONE,
                      BUSY => #BUSY,
                      ERROR => #ERROR,
                      STATUS => #STATUS);
   #_odk_internal_Last_BUSY := #BUSY;
   //
   // DO NOT CHANGE !!
   // This is an automatic generated block by the
   // SIMATIC ODK 1500S V2.0
   // DO NOT CHANGE ABOVE OF THIS LINE !!
   //
END_FUNCTION_BLOCK

FUNCTION "FFT_LoadUnload" : Void   // FC1, FBD
{ S7_Optimized_Access := 'TRUE' }
VERSION : 0.1
   VAR_TEMP   // added for the SCL form of the ladder/FBD networks
      _w1 : Bool;
      _w2 : Bool;
      _w3 : Bool;
      _w4 : Bool;
      _w5 : Bool;
   END_VAR
BEGIN

REGION Network 1
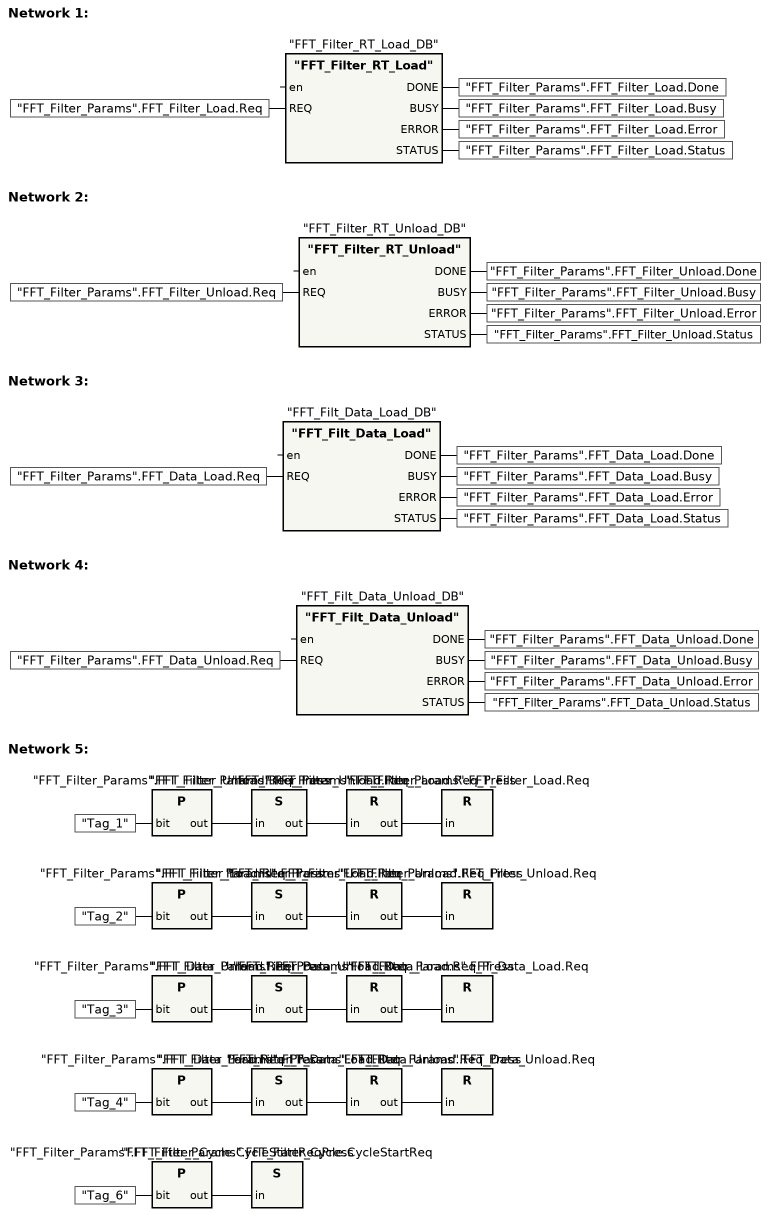
   "FFT_Filter_RT_Load_DB"(REQ := "FFT_Filter_Params".FFT_Filter_Load.Req,   // "FFT_Filter_RT_Load"
                           DONE => "FFT_Filter_Params".FFT_Filter_Load.Done,
                           BUSY => "FFT_Filter_Params".FFT_Filter_Load.Busy,
                           ERROR => "FFT_Filter_Params".FFT_Filter_Load.Error,
                           STATUS => "FFT_Filter_Params".FFT_Filter_Load.Status);
END_REGION

REGION Network 2
   "FFT_Filter_RT_Unload_DB"(REQ := "FFT_Filter_Params".FFT_Filter_Unload.Req,   // "FFT_Filter_RT_Unload"
                           DONE => "FFT_Filter_Params".FFT_Filter_Unload.Done,
                           BUSY => "FFT_Filter_Params".FFT_Filter_Unload.Busy,
                           ERROR => "FFT_Filter_Params".FFT_Filter_Unload.Error,
                           STATUS => "FFT_Filter_Params".FFT_Filter_Unload.Status);
END_REGION

REGION Network 3
   "FFT_Filt_Data_Load_DB"(REQ := "FFT_Filter_Params".FFT_Data_Load.Req,   // "FFT_Filt_Data_Load"
                           DONE => "FFT_Filter_Params".FFT_Data_Load.Done,
                           BUSY => "FFT_Filter_Params".FFT_Data_Load.Busy,
                           ERROR => "FFT_Filter_Params".FFT_Data_Load.Error,
                           STATUS => "FFT_Filter_Params".FFT_Data_Load.Status);
END_REGION

REGION Network 4
   "FFT_Filt_Data_Unload_DB"(REQ := "FFT_Filter_Params".FFT_Data_Unload.Req,   // "FFT_Filt_Data_Unload"
                           DONE => "FFT_Filter_Params".FFT_Data_Unload.Done,
                           BUSY => "FFT_Filter_Params".FFT_Data_Unload.Busy,
                           ERROR => "FFT_Filter_Params".FFT_Data_Unload.Error,
                           STATUS => "FFT_Filter_Params".FFT_Data_Unload.Status);
END_REGION

REGION Network 5
   #_w1 := "FFT_Filter_Params".FFT_Filter_Unload.Req_Press AND NOT "Tag_1";   // rising edge of "FFT_Filter_Params".FFT_Filter_Unload.Req_Press
   "Tag_1" := "FFT_Filter_Params".FFT_Filter_Unload.Req_Press;
   IF #_w1 THEN
       "FFT_Filter_Params".FFT_Filter_Unload.Req := TRUE;
       "FFT_Filter_Params".FFT_Filter_Load.Req_Press := FALSE;
       "FFT_Filter_Params".FFT_Filter_Load.Req := FALSE;
   END_IF;
   #_w2 := "FFT_Filter_Params".FFT_Filter_Load.Req_Press AND NOT "Tag_2";   // rising edge of "FFT_Filter_Params".FFT_Filter_Load.Req_Press
   "Tag_2" := "FFT_Filter_Params".FFT_Filter_Load.Req_Press;
   IF #_w2 THEN
       "FFT_Filter_Params".FFT_Filter_Load.Req := TRUE;
       "FFT_Filter_Params".FFT_Filter_Unload.Req_Press := FALSE;
       "FFT_Filter_Params".FFT_Filter_Unload.Req := FALSE;
   END_IF;
   #_w3 := "FFT_Filter_Params".FFT_Data_Unload.Req_Press AND NOT "Tag_3";   // rising edge of "FFT_Filter_Params".FFT_Data_Unload.Req_Press
   "Tag_3" := "FFT_Filter_Params".FFT_Data_Unload.Req_Press;
   IF #_w3 THEN
       "FFT_Filter_Params".FFT_Data_Unload.Req := TRUE;
       "FFT_Filter_Params".FFT_Data_Load.Req_Press := FALSE;
       "FFT_Filter_Params".FFT_Data_Load.Req := FALSE;
   END_IF;
   #_w4 := "FFT_Filter_Params".FFT_Data_Load.Req_Press AND NOT "Tag_4";   // rising edge of "FFT_Filter_Params".FFT_Data_Load.Req_Press
   "Tag_4" := "FFT_Filter_Params".FFT_Data_Load.Req_Press;
   IF #_w4 THEN
       "FFT_Filter_Params".FFT_Data_Load.Req := TRUE;
       "FFT_Filter_Params".FFT_Data_Unload.Req_Press := FALSE;
       "FFT_Filter_Params".FFT_Data_Unload.Req := FALSE;
   END_IF;
   #_w5 := "FFT_Filter_Params".FFT_Filter_Cycle.CycleStartReqPress AND NOT "Tag_6";   // rising edge of "FFT_Filter_Params".FFT_Filter_Cycle.CycleStartReqPress
   "Tag_6" := "FFT_Filter_Params".FFT_Filter_Cycle.CycleStartReqPress;
   IF #_w5 THEN "FFT_Filter_Params".FFT_Filter_Cycle.CycleStartReq := TRUE; END_IF;
END_REGION
END_FUNCTION

FUNCTION "FFT_Cycle" : Void   // FC2, FBD
{ S7_Optimized_Access := 'TRUE' }
VERSION : 0.1
   VAR_TEMP   // added for the SCL form of the ladder/FBD networks
      _w1 : Bool;
   END_VAR
BEGIN

REGION Network 1
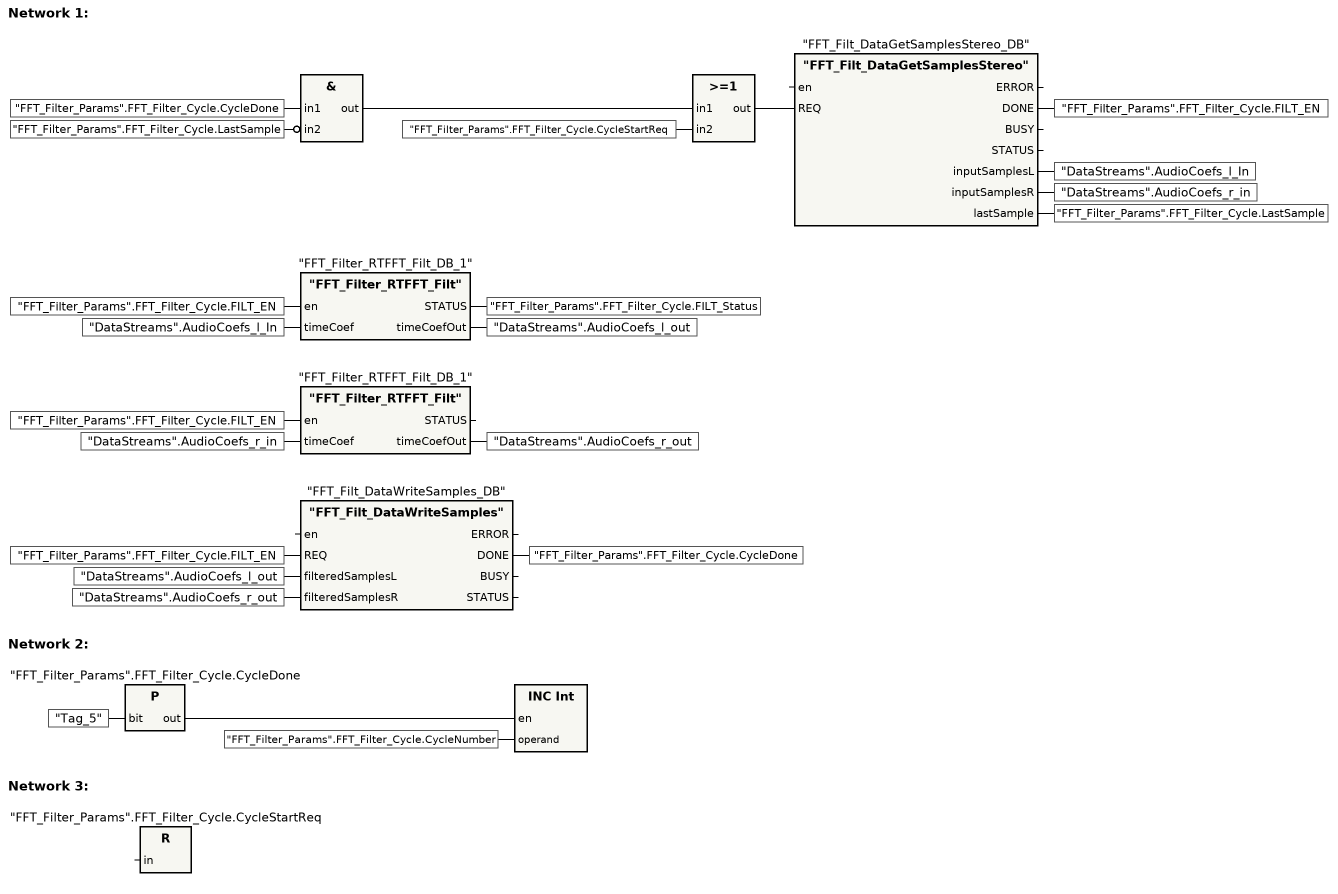
   "FFT_Filt_DataGetSamplesStereo_DB"(REQ := ("FFT_Filter_Params".FFT_Filter_Cycle.CycleDone AND NOT "FFT_Filter_Params".FFT_Filter_Cycle.LastSample) OR "FFT_Filter_Params".FFT_Filter_Cycle.CycleStartReq,   // "FFT_Filt_DataGetSamplesStereo"
                           DONE => "FFT_Filter_Params".FFT_Filter_Cycle.FILT_EN,
                           inputSamplesL => "DataStreams".AudioCoefs_l_In,
                           inputSamplesR => "DataStreams".AudioCoefs_r_in,
                           lastSample => "FFT_Filter_Params".FFT_Filter_Cycle.LastSample);
   IF "FFT_Filter_Params".FFT_Filter_Cycle.FILT_EN THEN
       "FFT_Filter_RTFFT_Filt_DB_1"(timeCoef := "DataStreams".AudioCoefs_l_In,   // "FFT_Filter_RTFFT_Filt"
                               STATUS => "FFT_Filter_Params".FFT_Filter_Cycle.FILT_Status,
                               timeCoefOut => "DataStreams".AudioCoefs_l_out);
   END_IF;
   IF "FFT_Filter_Params".FFT_Filter_Cycle.FILT_EN THEN
       "FFT_Filter_RTFFT_Filt_DB_1"(timeCoef := "DataStreams".AudioCoefs_r_in,   // "FFT_Filter_RTFFT_Filt"
                               timeCoefOut => "DataStreams".AudioCoefs_r_out);
   END_IF;
   "FFT_Filt_DataWriteSamples_DB"(REQ := "FFT_Filter_Params".FFT_Filter_Cycle.FILT_EN,   // "FFT_Filt_DataWriteSamples"
                           filteredSamplesL := "DataStreams".AudioCoefs_l_out,
                           filteredSamplesR := "DataStreams".AudioCoefs_r_out,
                           DONE => "FFT_Filter_Params".FFT_Filter_Cycle.CycleDone);
END_REGION

REGION Network 2
   #_w1 := "FFT_Filter_Params".FFT_Filter_Cycle.CycleDone AND NOT "Tag_5";   // rising edge of "FFT_Filter_Params".FFT_Filter_Cycle.CycleDone
   "Tag_5" := "FFT_Filter_Params".FFT_Filter_Cycle.CycleDone;
   IF #_w1 THEN
       "FFT_Filter_Params".FFT_Filter_Cycle.CycleNumber := "FFT_Filter_Params".FFT_Filter_Cycle.CycleNumber + 1;
   END_IF;
END_REGION

REGION Network 3
   "FFT_Filter_Params".FFT_Filter_Cycle.CycleStartReq := FALSE;
END_REGION
END_FUNCTION

ORGANIZATION_BLOCK "Main"   // OB1, LAD, ProgramCycle
TITLE = "Main Program Sweep (Cycle)"
{ S7_Optimized_Access := 'TRUE' }
VERSION : 0.1
   VAR_INPUT
      Initial_Call : Bool;   // Initial call of this OB
      Remanence : Bool;   // =True, if remanent data are available
   END_VAR
BEGIN

REGION Network 1
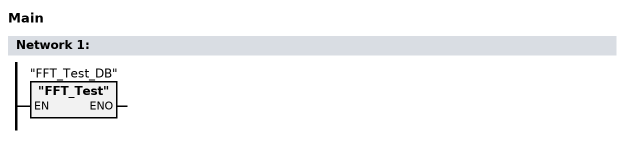
   RUNG wire#powerrail
      "FFT_Test_DB"()
   END_RUNG
   // the same network as SCL:
   "FFT_Test_DB"();   // "FFT_Test"
END_REGION
END_ORGANIZATION_BLOCK

(* ===== HMI "HMI_RT_1" =====
system functions are stored by id; their names below are inferred from use
connection "HMI_Connection_1": ETHERNET, SMART_S7_1500_OMS

HMI tags "Default tag table"
   "FFT_Filter_Params_FFT_Filter_Load_Status" : Int = PLC FFT_Filter_Params.FFT_Filter_Load.Status, 100 ms
   "FFT_Filter_Params_FFT_Filter_Load_Done" : Bool = PLC FFT_Filter_Params.FFT_Filter_Load.Done, 100 ms
   "FFT_Filter_Params_FFT_Filter_Load_Busy" : Bool = PLC FFT_Filter_Params.FFT_Filter_Load.Busy, 100 ms
   "FFT_Filter_Params_FFT_Filter_Load_Error" : Bool = PLC FFT_Filter_Params.FFT_Filter_Load.Error, 100 ms
   "FFT_Filter_Params_FFT_Filter_Load_Req" : Bool = PLC FFT_Filter_Params.FFT_Filter_Load.Req, 100 ms
   "FFT_Filter_Params_FFT_Filter_Unload_Req" : Bool = PLC FFT_Filter_Params.FFT_Filter_Unload.Req, 100 ms
   "FFT_Filter_Params_FFT_Filter_Unload_Error" : Bool = PLC FFT_Filter_Params.FFT_Filter_Unload.Error, 100 ms
   "FFT_Filter_Params_FFT_Filter_Unload_Busy" : Bool = PLC FFT_Filter_Params.FFT_Filter_Unload.Busy, 100 ms
   "FFT_Filter_Params_FFT_Filter_Unload_Done" : Bool = PLC FFT_Filter_Params.FFT_Filter_Unload.Done, 100 ms
   "FFT_Filter_Params_FFT_Filter_Unload_Status" : Int = PLC FFT_Filter_Params.FFT_Filter_Unload.Status, 100 ms
   "FFT_Filter_Params_FFT_Filter_Load_Req_Press" : Bool = PLC FFT_Filter_Params.FFT_Filter_Load.Req_Press, 100 ms
   "FFT_Filter_Params_FFT_Filter_Unload_Req_Press" : Bool = PLC FFT_Filter_Params.FFT_Filter_Unload.Req_Press, 100 ms
   "FFT_Filter_Params_FFT_Filter_Cycle_FILT_Status" : Int = PLC FFT_Filter_Params.FFT_Filter_Cycle.FILT_Status, 100 ms
   "FFT_Filter_Params_FFT_Filter_Cycle_FILT_EN" : Bool = PLC FFT_Filter_Params.FFT_Filter_Cycle.FILT_EN, 100 ms
   "FFT_Filter_Params_FFT_Data_Load_Status" : Int = PLC FFT_Filter_Params.FFT_Data_Load.Status, 100 ms
   "FFT_Filter_Params_FFT_Data_Load_Done" : Bool = PLC FFT_Filter_Params.FFT_Data_Load.Done, 100 ms
   "FFT_Filter_Params_FFT_Data_Load_Busy" : Bool = PLC FFT_Filter_Params.FFT_Data_Load.Busy, 100 ms
   "FFT_Filter_Params_FFT_Data_Load_Error" : Bool = PLC FFT_Filter_Params.FFT_Data_Load.Error, 100 ms
   "FFT_Filter_Params_FFT_Data_Load_Req" : Bool = PLC FFT_Filter_Params.FFT_Data_Load.Req, 100 ms
   "FFT_Filter_Params_FFT_Data_Unload_Status" : Int = PLC FFT_Filter_Params.FFT_Data_Unload.Status, 100 ms
   "FFT_Filter_Params_FFT_Data_Unload_Done" : Bool = PLC FFT_Filter_Params.FFT_Data_Unload.Done, 100 ms
   "FFT_Filter_Params_FFT_Data_Unload_Busy" : Bool = PLC FFT_Filter_Params.FFT_Data_Unload.Busy, 100 ms
   "FFT_Filter_Params_FFT_Data_Unload_Error" : Bool = PLC FFT_Filter_Params.FFT_Data_Unload.Error, 100 ms
   "FFT_Filter_Params_FFT_Data_Unload_Req" : Bool = PLC FFT_Filter_Params.FFT_Data_Unload.Req, 100 ms
   "FFT_Filter_Params_FFT_Data_Load_Req_Press" : Bool = PLC FFT_Filter_Params.FFT_Data_Load.Req_Press, 100 ms
   "FFT_Filter_Params_FFT_Data_Unload_Req_Press" : Bool = PLC FFT_Filter_Params.FFT_Data_Unload.Req_Press, 100 ms
   "FFT_Filter_Params_FFT_Filter_Cycle_CycleNumber" : Int = PLC FFT_Filter_Params.FFT_Filter_Cycle.CycleNumber, 100 ms
   "FFT_Filter_Params_FFT_Filter_Cycle_LastSample" : Bool = PLC FFT_Filter_Params.FFT_Filter_Cycle.LastSample, 100 ms
   "FFT_Filter_Params_FFT_Filter_Cycle_CycleStartReqPress" : Bool = PLC FFT_Filter_Params.FFT_Filter_Cycle.CycleStartReqPress, 100 ms

screen "Screen_1" 800x480
   IOField "I/O field_1" at 182,29 size 70x32; FormatPattern FFFF
      ProcessValue <- "FFT_Filter_Params_FFT_Filter_Load_Status"
   IOField "I/O field_2" at 182,61 size 70x32; FormatPattern 1
      ProcessValue <- "FFT_Filter_Params_FFT_Filter_Load_Done"
   TextField "Text field_1" at 23,32 size 143x23; Text 'Filter load status'
   TextField "Text field_2" at 23,64 size 133x23; Text 'Filter load done'
   TextField "Text field_3" at 23,96 size 130x23; Text 'Filter load busy'
   TextField "Text field_4" at 23,128 size 134x23; Text 'Filter load error'
   IOField "I/O field_3" at 182,93 size 70x32; FormatPattern 1
      ProcessValue <- "FFT_Filter_Params_FFT_Filter_Load_Busy"
   IOField "I/O field_4" at 182,125 size 70x32; FormatPattern 1
      ProcessValue <- "FFT_Filter_Params_FFT_Filter_Load_Error"
   Button "Button_1" at 23,201 size 96x32; TextOff 'Load'
      on Release: SetBit("FFT_Filter_Params_FFT_Filter_Load_Req_Press")
   TextField "Text field_5" at 23,160 size 120x23; Text 'Filter load req'
   IOField "I/O field_5" at 182,157 size 70x32; FormatPattern 1
      ProcessValue <- "FFT_Filter_Params_FFT_Filter_Load_Req"
   IOField "I/O field_6" at 464,29 size 70x32; FormatPattern FFFF
      ProcessValue <- "FFT_Filter_Params_FFT_Filter_Unload_Status"
   IOField "I/O field_7" at 464,61 size 70x32; FormatPattern 1
      ProcessValue <- "FFT_Filter_Params_FFT_Filter_Unload_Done"
   TextField "Text field_6" at 305,32 size 163x23; Text 'Filter unload status'
   TextField "Text field_7" at 305,64 size 153x23; Text 'Filter unload done'
   TextField "Text field_8" at 305,96 size 150x23; Text 'Filter unload busy'
   TextField "Text field_9" at 305,128 size 154x23; Text 'Filter unload error'
   IOField "I/O field_8" at 464,93 size 70x32; FormatPattern 1
      ProcessValue <- "FFT_Filter_Params_FFT_Filter_Unload_Busy"
   IOField "I/O field_9" at 464,125 size 70x32; FormatPattern 1
      ProcessValue <- "FFT_Filter_Params_FFT_Filter_Unload_Error"
   Button "Button_2" at 305,201 size 96x32; TextOff 'Unload'
      on Release: SetBit("FFT_Filter_Params_FFT_Filter_Unload_Req_Press")
   TextField "Text field_10" at 305,160 size 140x23; Text 'Filter unload req'
   IOField "I/O field_10" at 464,157 size 70x32; FormatPattern 1
      ProcessValue <- "FFT_Filter_Params_FFT_Filter_Unload_Req"
   IOField "I/O field_11" at 719,29 size 70x32; FormatPattern FFFF
      ProcessValue <- "FFT_Filter_Params_FFT_Filter_Cycle_FILT_Status"
   IOField "I/O field_12" at 719,61 size 70x32; FormatPattern 1
      ProcessValue <- "FFT_Filter_Params_FFT_Filter_Cycle_FILT_EN"
   TextField "Text field_11" at 560,32 size 103x23; Text 'Filter status'
   TextField "Text field_12" at 560,64 size 118x23; Text 'Filter enabled'
   IOField "I/O field_13" at 182,258 size 70x32; FormatPattern FFFF
      ProcessValue <- "FFT_Filter_Params_FFT_Data_Load_Status"
   IOField "I/O field_14" at 182,290 size 70x32; FormatPattern 1
      ProcessValue <- "FFT_Filter_Params_FFT_Data_Load_Done"
   TextField "Text field_13" at 23,261 size 139x23; Text 'Data load status'
   TextField "Text field_14" at 23,293 size 129x23; Text 'Data load done'
   TextField "Text field_15" at 23,325 size 126x23; Text 'Data load busy'
   TextField "Text field_16" at 23,357 size 130x23; Text 'Data load error'
   IOField "I/O field_15" at 182,322 size 70x32; FormatPattern 1
      ProcessValue <- "FFT_Filter_Params_FFT_Data_Load_Busy"
   IOField "I/O field_16" at 182,354 size 70x32; FormatPattern 1
      ProcessValue <- "FFT_Filter_Params_FFT_Data_Load_Error"
   Button "Button_3" at 23,430 size 96x32; TextOff 'Load'
      on Release: SetBit("FFT_Filter_Params_FFT_Data_Load_Req_Press")
   TextField "Text field_17" at 23,389 size 116x23; Text 'Data load req'
   IOField "I/O field_17" at 182,386 size 70x32; FormatPattern 1
      ProcessValue <- "FFT_Filter_Params_FFT_Data_Load_Req"
   IOField "I/O field_18" at 464,258 size 70x32; FormatPattern FFFF
      ProcessValue <- "FFT_Filter_Params_FFT_Data_Unload_Status"
   IOField "I/O field_19" at 464,290 size 70x32; FormatPattern 1
      ProcessValue <- "FFT_Filter_Params_FFT_Data_Unload_Done"
   TextField "Text field_18" at 305,261 size 159x23; Text 'Data unload status'
   TextField "Text field_19" at 305,293 size 149x23; Text 'Data unload done'
   TextField "Text field_20" at 305,325 size 146x23; Text 'Data unload busy'
   TextField "Text field_21" at 305,357 size 150x23; Text 'Data unload error'
   IOField "I/O field_20" at 464,322 size 70x32; FormatPattern 1
      ProcessValue <- "FFT_Filter_Params_FFT_Data_Unload_Busy"
   IOField "I/O field_21" at 464,354 size 70x32; FormatPattern 1
      ProcessValue <- "FFT_Filter_Params_FFT_Data_Unload_Error"
   Button "Button_4" at 305,430 size 96x32; TextOff 'Unload'
      on Release: SetBit("FFT_Filter_Params_FFT_Data_Unload_Req_Press")
   TextField "Text field_22" at 305,389 size 136x23; Text 'Data unload req'
   IOField "I/O field_22" at 464,386 size 70x32; FormatPattern 1
      ProcessValue <- "FFT_Filter_Params_FFT_Data_Unload_Req"
   IOField "I/O field_23" at 719,257 size 70x32; FormatPattern FFFF
      ProcessValue <- "FFT_Filter_Params_FFT_Filter_Cycle_CycleNumber"
   IOField "I/O field_24" at 719,289 size 70x32; FormatPattern 1
      ProcessValue <- "FFT_Filter_Params_FFT_Filter_Cycle_LastSample"
   TextField "Text field_23" at 560,260 size 117x23; Text 'Cycle Number'
   TextField "Text field_24" at 560,292 size 104x23; Text 'Last Sample'
   Button "Button_5" at 560,329 size 96x32; TextOff 'Start'
      on Release: SetBit("FFT_Filter_Params_FFT_Filter_Cycle_CycleStartReqPress")

screen "Screen_2" 800x480
   SysDiagControl "System diagnostics view_1" at 0,0 size 747x479
*)